FUNCTION_BLOCK FB_ControlSignal
VAR_INPUT
	fUFF : LREAL;
	fPID : LREAL;
	bEnableU : BOOL;
	fQMaxUp 	: LREAL; // Needs to be positive (22)
	fQMaxDown 	: LREAL; // Needs to be positive (15)
	fDeadUp		: LREAL; // Needs to be positive (0.155)
	fDeadDown 	: LREAL; // Needs to be positive (0.18)
END_VAR
VAR_OUTPUT
	fU : LREAL;
END_VAR
VAR
	fSignalMax : LREAL := 1.0;
	fSignalMin : LREAL := -1.0;
	fUTemp : LREAL;
	fUTemp2 : LREAL;
	fUMax : LREAL := 0.9;
END_VAR

IF bEnableU THEN
	fUTemp := fUFF - fPID;
	
// Deadband compensation
IF fUTemp <= 0.0 THEN	
	IF fUTemp < -fUMax THEN // Upwards
		fUTemp2 := -fUMax;
	
	ELSIF fUTemp > -fDeadUp THEN
		fUTemp2 := -fDeadUp;
	ELSE
		fUTemp2 := fUTemp - fDeadUp;
	END_IF

ELSIF fUTemp > 0.0 THEN
	
	IF fUTemp > fUMax THEN // Downwards
		fUTemp2 := fUMax;
	
	ELSIF fUTemp < fDeadDown THEN
		fUTemp2 := fDeadDown;
	ELSE
		fUTemp2 := fUTemp + fDeadDown;
	END_IF
END_IF
	
	IF fUTemp2 >= fSignalMax THEN
		fU := fSignalMax;
	ELSIF fUTemp2 <= fSignalMin THEN
		fU := fSignalMin;
	ELSE
		fU := fUTemp2;
	END_IF
	
ELSE
	fU := 0.0;
END_IF

END_FUNCTION_BLOCK

(* stored: Version 1.1.0.1, ProductVersion 3.1.4024.12
   POU FB_ControlSignal: Id {5ec98e7b-f91c-4803-9df2-1eb6eb99ed16}, SpecialFunc None *)
